ABB RAPID module: 001066C2

MODULE CalibData
    PERS tooldata MoldGripper:=[TRUE,[[-10.5,0,100],[1,0,0,0]],[1.873,[-1.681,0,-0.205],[1,0,0,0],0.002877912,0.002365912,0.002366511]];
    TASK PERS wobjdata BaseMolds:=[FALSE,TRUE,"",[[1700,200,1200],[0.5,-0.5,0.5,0.5]],[[0,0,0],[1,0,0,0]]];
    CONST robtarget BaseL_1:=[[-184.986,250,-10],[1,0,0,0],[-1,0,-2,0],[9E+09,9E+09,9E+09,9E+09,9E+09,9E+09]];
    CONST robtarget BaseL_2:=[[-184.986,250,85],[1,0,0,0],[0,1,-2,0],[9E+09,9E+09,9E+09,9E+09,9E+09,9E+09]];
    CONST robtarget BaseL_3:=[[-204.986,250,85],[1,0,0,0],[0,1,-2,0],[9E+09,9E+09,9E+09,9E+09,9E+09,9E+09]];
    CONST robtarget BaseL_4:=[[-224.986,250,85],[1,0,0,0],[0,1,-2,0],[9E+09,9E+09,9E+09,9E+09,9E+09,9E+09]];
    CONST robtarget BaseL_5:=[[-324.986,250,85],[1,0,0,0],[0,0,-1,0],[9E+09,9E+09,9E+09,9E+09,9E+09,9E+09]];
    CONST robtarget BaseL_6:=[[-324.986,250,-15],[1,0,0,0],[-1,1,-1,0],[9E+09,9E+09,9E+09,9E+09,9E+09,9E+09]];
    CONST robtarget BaseL_7:=[[-324.986,1250,-15],[1,0,0,0],[-1,1,-1,0],[9E+09,9E+09,9E+09,9E+09,9E+09,9E+09]];

    CONST robtarget BaseR_1:=[[-184.986,250,-390],[0,1,0,0],[0,-1,1,0],[9E+09,9E+09,9E+09,9E+09,9E+09,9E+09]];
    CONST robtarget BaseR_2:=[[-184.986,250,-485],[0,1,0,0],[-1,-2,1,0],[9E+09,9E+09,9E+09,9E+09,9E+09,9E+09]];
    CONST robtarget BaseR_3:=[[-204.986,250,-485],[0,1,0,0],[-1,-2,1,0],[9E+09,9E+09,9E+09,9E+09,9E+09,9E+09]];
    CONST robtarget BaseR_4:=[[-224.986,250,-485],[0,1,0,0],[-1,-2,1,0],[9E+09,9E+09,9E+09,9E+09,9E+09,9E+09]];
    CONST robtarget BaseR_5:=[[-324.986,250,-485],[0,1,0,0],[-1,-1,0,0],[9E+09,9E+09,9E+09,9E+09,9E+09,9E+09]];
    CONST robtarget BaseR_6:=[[-324.986,250,-385],[0,1,0,0],[0,-2,0,0],[9E+09,9E+09,9E+09,9E+09,9E+09,9E+09]];
    CONST robtarget BaseR_7:=[[-324.986,1250,-385],[0,1,0,0],[0,-2,0,0],[9E+09,9E+09,9E+09,9E+09,9E+09,9E+09]];

    CONST robtarget Home:=[[-175,1200,-200],[0.707106781,0.707106781,0,0],[0,0,0,0],[9E+09,9E+09,9E+09,9E+09,9E+09,9E+09]];

    TASK PERS wobjdata LeftMoldStore:=[FALSE,TRUE,"",[[250,1550,1500],[0.5,-0.5,0.5,0.5]],[[0,0,0],[1,0,0,0]]];
    CONST robtarget BlackL_1:=[[215.014,250,-110],[1,0,0,0],[1,-1,0,1],[9E+09,9E+09,9E+09,9E+09,9E+09,9E+09]];
    CONST robtarget BlackL_2:=[[215.014,250,-10],[1,0,0,0],[1,-1,0,1],[9E+09,9E+09,9E+09,9E+09,9E+09,9E+09]];
    CONST robtarget BlackL_3:=[[215.014,250,85],[1,0,0,0],[1,-1,0,1],[9E+09,9E+09,9E+09,9E+09,9E+09,9E+09]];
    CONST robtarget BlackL_4:=[[195.014,250,85],[1,0,0,0],[1,-1,0,1],[9E+09,9E+09,9E+09,9E+09,9E+09,9E+09]];
    CONST robtarget BlackL_5:=[[175.014,250,85],[1,0,0,0],[1,-1,0,1],[9E+09,9E+09,9E+09,9E+09,9E+09,9E+09]];
    CONST robtarget BlackL_6:=[[175.014,250,-315],[1,0,0,0],[1,-1,0,1],[9E+09,9E+09,9E+09,9E+09,9E+09,9E+09]];
    CONST robtarget RedL_1:=[[715.014,250,-110],[1,0,0,0],[1,-1,0,1],[9E+09,9E+09,9E+09,9E+09,9E+09,9E+09]];
    CONST robtarget RedL_2:=[[715.014,250,-10],[1,0,0,0],[1,-1,0,1],[9E+09,9E+09,9E+09,9E+09,9E+09,9E+09]];
    CONST robtarget RedL_3:=[[715.014,250,85],[1,0,0,0],[1,-1,0,1],[9E+09,9E+09,9E+09,9E+09,9E+09,9E+09]];
    CONST robtarget RedL_4:=[[695.014,250,85],[1,0,0,0],[1,-1,0,1],[9E+09,9E+09,9E+09,9E+09,9E+09,9E+09]];
    CONST robtarget RedL_5:=[[675.014,250,85],[1,0,0,0],[1,-1,0,1],[9E+09,9E+09,9E+09,9E+09,9E+09,9E+09]];
    CONST robtarget RedL_6:=[[675.014,250,-315],[1,0,0,0],[1,-1,0,1],[9E+09,9E+09,9E+09,9E+09,9E+09,9E+09]];
    CONST robtarget BlueL_1:=[[1215.014,250,-110],[1,0,0,0],[1,0,0,1],[9E+09,9E+09,9E+09,9E+09,9E+09,9E+09]];
    CONST robtarget BlueL_2:=[[1215.014,250,-10],[1,0,0,0],[1,0,0,1],[9E+09,9E+09,9E+09,9E+09,9E+09,9E+09]];
    CONST robtarget BlueL_3:=[[1215.014,250,85],[1,0,0,0],[1,0,0,1],[9E+09,9E+09,9E+09,9E+09,9E+09,9E+09]];
    CONST robtarget BlueL_5:=[[1175.014,250,85],[1,0,0,0],[1,0,0,1],[9E+09,9E+09,9E+09,9E+09,9E+09,9E+09]];
    CONST robtarget BlueL_4:=[[1195.014,250,85],[1,0,0,0],[1,0,0,1],[9E+09,9E+09,9E+09,9E+09,9E+09,9E+09]];
    CONST robtarget BlueL_6:=[[1175.014,250,-315],[1,0,0,0],[1,0,0,1],[9E+09,9E+09,9E+09,9E+09,9E+09,9E+09]];

    CONST robtarget LeftHome:=[[175.014,250,-865],[1,0,0,0],[1,0,-1,0],[9E+09,9E+09,9E+09,9E+09,9E+09,9E+09]];

    TASK PERS wobjdata RightMoldStore:=[FALSE,TRUE,"",[[-250,-1550,1500],[0.5,0.5,0.5,-0.5]],[[0,0,0],[1,0,0,0]]];

    CONST robtarget BlackR_1:=[[215.014,250,-110],[1,0,0,0],[-1,0,-1,1],[9E+09,9E+09,9E+09,9E+09,9E+09,9E+09]];
    CONST robtarget BlackR_2:=[[215.014,250,-10],[1,0,0,0],[-1,-1,0,1],[9E+09,9E+09,9E+09,9E+09,9E+09,9E+09]];
    CONST robtarget BlackR_3:=[[215.014,250,85],[1,0,0,0],[-1,-1,0,1],[9E+09,9E+09,9E+09,9E+09,9E+09,9E+09]];
    CONST robtarget BlackR_4:=[[195.014,250,85],[1,0,0,0],[-1,-1,0,1],[9E+09,9E+09,9E+09,9E+09,9E+09,9E+09]];
    CONST robtarget BlackR_5:=[[175.014,250,85],[1,0,0,0],[-1,-1,0,1],[9E+09,9E+09,9E+09,9E+09,9E+09,9E+09]];
    CONST robtarget BlackR_6:=[[175.014,250,-315],[1,0,0,0],[-1,-1,0,1],[9E+09,9E+09,9E+09,9E+09,9E+09,9E+09]];
    CONST robtarget RedR_1:=[[715.014,250,-110],[1,0,0,0],[-1,0,-1,1],[9E+09,9E+09,9E+09,9E+09,9E+09,9E+09]];
    CONST robtarget RedR_2:=[[715.014,250,-10],[1,0,0,0],[-1,-1,0,1],[9E+09,9E+09,9E+09,9E+09,9E+09,9E+09]];
    CONST robtarget RedR_3:=[[715.014,250,85],[1,0,0,0],[-1,-1,0,1],[9E+09,9E+09,9E+09,9E+09,9E+09,9E+09]];
    CONST robtarget RedR_4:=[[695.014,250,85],[1,0,0,0],[-1,-1,0,1],[9E+09,9E+09,9E+09,9E+09,9E+09,9E+09]];
    CONST robtarget RedR_5:=[[675.014,250,85],[1,0,0,0],[-1,0,-1,1],[9E+09,9E+09,9E+09,9E+09,9E+09,9E+09]];
    CONST robtarget RedR_6:=[[675.014,250,-315],[1,0,0,0],[-1,0,-1,1],[9E+09,9E+09,9E+09,9E+09,9E+09,9E+09]];
    CONST robtarget BlueR_1:=[[1215.014,250,-110],[1,0,0,0],[-1,0,-1,1],[9E+09,9E+09,9E+09,9E+09,9E+09,9E+09]];
    CONST robtarget BlueR_2:=[[1215.014,250,-10],[1,0,0,0],[-1,0,0,1],[9E+09,9E+09,9E+09,9E+09,9E+09,9E+09]];
    CONST robtarget BlueR_3:=[[1215.014,250,85],[1,0,0,0],[-1,0,0,1],[9E+09,9E+09,9E+09,9E+09,9E+09,9E+09]];
    CONST robtarget BlueR_4:=[[1195.014,250,85],[1,0,0,0],[-1,0,0,1],[9E+09,9E+09,9E+09,9E+09,9E+09,9E+09]];
    CONST robtarget BlueR_5:=[[1175.014,250,85],[1,0,0,0],[-1,0,-1,1],[9E+09,9E+09,9E+09,9E+09,9E+09,9E+09]];
    CONST robtarget BlueR_6:=[[1175.014,250,-315],[1,0,0,0],[-1,0,0,1],[9E+09,9E+09,9E+09,9E+09,9E+09,9E+09]];

    CONST robtarget RightHome:=[[175.014,250,-765],[1,0,0,0],[-1,1,-2,1],[9E+09,9E+09,9E+09,9E+09,9E+09,9E+09]];

ENDMODULE
